# EPICS substitutions: lakeshore336App/Db/lakeshore336_curve.substitutions
file "lakeshore336_curve.template"
{
	pattern { CurveType }

	{  File }
	{  ""   }
}
